{attribute 'GeneratedUsingTerminal: KL2641-0001'}
{attribute addProperty BoxType "KL2641-0001"}
{attribute addProperty Id "Manual_StateAT %I*BOOL0ReservedAT %I*BOOL0OutputAT %Q*BOOL0"}
{attribute addProperty CRC "3208012237"}
{attribute addProperty Size "0"}
TYPE Channel_BF3661CD :
STRUCT
	{attribute addProperty Name "Manual_State"}
	Manual_State AT %I* : BOOL;
	{attribute addProperty Name "Reserved"}
	Reserved AT %I* : BOOL;
	{attribute addProperty Name "Output"}
	Output AT %Q* : BOOL;
END_STRUCT
END_TYPE

(* stored: Version 1.2.0.0, ProductVersion 3.1.4024.9
   DUT Channel_BF3661CD: Id {e3018545-4059-4b41-b594-d8e0606411ba} *)
